FUNCTION FB_SPS_zu_Nativ_lin : REAL
VAR_INPUT
	Input: INPUT_VAR;
	
END_VAR
VAR

END_VAR

FB_SPS_zu_Nativ_lin:=Input.REAL_PARA_M*input.INT_VAR_Input+input.REAL_PARA_C;

END_FUNCTION

(* stored: Version 1.1.0.1, ProductVersion 3.1.4018.5
   POU FB_SPS_zu_Nativ_lin: Id {9bcdb250-b10f-4ae5-acb4-e1bcaada499c}, SpecialFunc None *)
